FUNCTION_BLOCK T_ModeManager IMPLEMENTS I_ModeManager
VAR
  _state : I_StateModule;
  _LogModeChanges : BOOL := TRUE;
  _CurrentMode : E_PMLUnitMode; //Current UnitMode of the module	
  _CommandedMode : E_PMLUnitMode; //Current Commanded UnitMode of the module

  PackModeManager : PML_UnitModeManager;
  CustomModes : PML_UnitModeConfig;
  LastModeCommand : E_PMLUnitMode;
  PMLModeLogger : FB_PackML_ModeLogger;
  LastMode : DINT;
  _ModeNames : ARRAY[0..31] OF STRING; // ('Production','Maintenance', 'Manual');
  ModeChangeRequested : BOOL;

  CurrentStrategy : I_PackMode := ProductionMode;
  ProductionMode : I_PackMode;
  MaintenanceMode : I_PackMode;
  ManualMode : I_PackMode;
  CustomPackModes : ARRAY[0..15] OF I_PackMode; // mobject ?
END_VAR

METHOD AddCustomPackMode : BOOL
VAR_INPUT
  index : UINT;
  newPackMode : I_PackMode;
END_VAR
custompackmodes[index] := newPackMode;
END_METHOD

METHOD AddPackModes : BOOL
VAR_INPUT
  prodMode : I_PackMode;
  maintMode : I_PackMode;
  manMode : I_PackMode;
END_VAR
ProductionMode := prodMode;
MaintenanceMode := maintMode;
ManualMode := manMode;
END_METHOD

METHOD PUBLIC AddStateModule
VAR_INPUT
  stateModule : I_StateModule;
END_VAR
_state := stateModule;
END_METHOD

METHOD PUBLIC ChangeMode
VAR_INPUT
  Mode : E_PMLUnitMode;
END_VAR
IF Mode <> _CommandedMode THEN
    _CommandedMode := Mode;
END_IF
END_METHOD

PROPERTY PUBLIC CommandedMode : E_PMLProtectedUnitMode
GET
CommandedMode := _CommandedMode;
END_GET
END_PROPERTY

PROPERTY CurrentMode : E_PMLProtectedUnitMode
GET
CurrentMode := _CurrentMode;
END_GET
END_PROPERTY

METHOD PUBLIC CyclicLogic
VAR_INPUT
END_VAR
ModeControl();
END_METHOD

METHOD FB_init : BOOL
VAR_INPUT
	bInitRetains : BOOL; // if TRUE, the retain variables are initialized (warm start / cold start)
	bInCopyCode : BOOL;  // if TRUE, the instance afterwards gets moved into the copy code (online change)
  stateModule : I_StateModule;
END_VAR
_state := stateModule;
END_METHOD

METHOD PRIVATE ListenForModeChange
VAR_INPUT
END_VAR

//On startup, Mode is invalid, set it to production
IF _CurrentMode = E_PMLUnitMode.ePMLUnitMode_Invalid THEN
    ModeChangeRequested := TRUE;
    _CommandedMode      := Parameters_PackML_Base.UNIT_MODE_DEFAULT;
    LastModeCommand := _CommandedMode;

    //If mode is valid and the command has changed, attempt to change modes
ELSIF _CommandedMode <> LastModeCommand THEN
    ModeChangeRequested               := TRUE;

    LastModeCommand := _CommandedMode;
END_IF
END_METHOD

PROPERTY PUBLIC LogModeChanges : BOOL
GET
LogModeChanges := _LogModeChanges;
END_GET
SET
_LogModeChanges := LogModeChanges;
END_SET
END_PROPERTY

METHOD PRIVATE ModeChange
VAR_INPUT
END_VAR

VAR
  SequenceState, DescendantSequenceState : UINT;
END_VAR
    //Handles mode changes based on ModeCommand and the state transition rules defined in the pre-defined protected modes or custom modes
    PackModeManager(bExecute     := TRUE,
                eModeCommand := _CommandedMode,
                eState       := _state.CurrentState,
                eModeStatus  => _CurrentMode);

        //If PackML mode has changed
        IF PackModeManager.eModeStatus <> LastMode THEN
            LastMode                := PackModeManager.eModeStatus;
            SequenceState           := 0;
            DescendantSequenceState := 0;

            //If state change logging is not suppressed
            IF _LogModeChanges THEN
                //PMLModeLogger(Alarms := PackMLAlarms, ModulePrefix := _Name, Mode := ModeManager.eModeStatus);
            END_IF

        END_IF

        // Reset mode control command
        PackModeManager(bExecute := FALSE);
        ModeChangeRequested := FALSE;
        
    IF PackModeManager.bError THEN
        //IF ReachedInitialDefaultStateAndMode THEN
        //    IF NOT PackMLAlarms[E_PackMLBase_Alarms.ModeCommandInvalid].bRaised THEN
        //        PackMLAlarms[E_PackMLBase_Alarms.ModeCommandInvalid].Raise(0);
        //    END_IF
        //END_IF

        // Reset mode control command
        PackModeManager(bExecute := FALSE);
        ModeChangeRequested := FALSE;
     END_IF
END_METHOD

METHOD PRIVATE ModeControl //Final ?
VAR
END_VAR
ListenForModeChange();

IF ModeChangeRequested THEN
    ModeChange();
END_IF
END_METHOD

PROPERTY PUBLIC  ModeNames : REFERENCE TO ARRAY[0..31] OF STRING
GET
ModeNames REF= _ModeNames;
END_GET
END_PROPERTY

END_FUNCTION_BLOCK

(* stored: Version 1.1.0.1, ProductVersion 3.1.4024.12
   POU T_ModeManager: Id {ea4887d2-59b6-4466-9a73-4e1ef78db5cc}, SpecialFunc None
   Folder Private: Id {5e3cd00c-f349-44a6-b04a-0f911deef120}
   Folder Properties: Id {62ed7422-cd3b-4ece-b766-f08a5786b32e}
   Folder Public: Id {63204732-e3ed-499c-a1cc-5d83bb8d3ea1}
   Method AddCustomPackMode: Id {6ea33754-fbd2-44c2-b121-20d3288e8049}
   Method AddPackModes: Id {85ef9fb9-fb0f-40b0-a83e-84ca52cbb7f9}
   Method AddStateModule: Id {21fe5c2d-7a9b-4ad5-84ff-7ae76830a6cd}
   Method ChangeMode: Id {bd04e302-796d-445f-9395-38f8b1c8f63e}
   Property CommandedMode: Id {e92ac6e2-3b07-41c3-9cac-aa4e0b94fdb1}
   Get Get: Id {c3433c3b-dcb6-45e1-b15a-0ce485f7e416}
   Property CurrentMode: Id {bb96f9bc-1fcf-4ca4-92d4-7395e019defd}
   Get Get: Id {91c66e1f-6a18-49bb-b03e-42a8637455f2}
   Method CyclicLogic: Id {0e92f0a6-71a1-4978-80c8-56ca48fef23c}
   Method FB_init: Id {bba8bd93-3ac1-495e-a997-963b53b268fd}
   Method ListenForModeChange: Id {e0d2514d-fec9-45cd-834c-1067f21c9d10}
   Property LogModeChanges: Id {b31cab9f-6f34-4e52-aa0b-dc94d5e9dd9a}
   Get Get: Id {7374b8d1-413d-4a11-b76e-8f1b8b163e74}
   Set Set: Id {27a04a66-2e65-4601-ad71-d45eda7902f4}
   Method ModeChange: Id {d05f0be5-01e9-43f5-8ab0-a0bdd61d255d}
   Method ModeControl: Id {b6127da8-0de3-408d-a711-2f3c4fe9482b}
   Property ModeNames: Id {e39c07a9-4860-45a1-a437-95f8bf6a1204}
   Get Get: Id {873d49e1-5c7c-48b4-a0a7-fef2bd7819e8} *)
